(* CODESYS project WaterGAState.export

Project tree, tasks and I/O mapping:
  data type GA_State
*)

// GA_State
//{attribute 'qualified_only'}
//{attribute 'strict'}
TYPE GA_State :
(
	S_Init,
	S_Ready,
	S_Busy
);
END_TYPE
